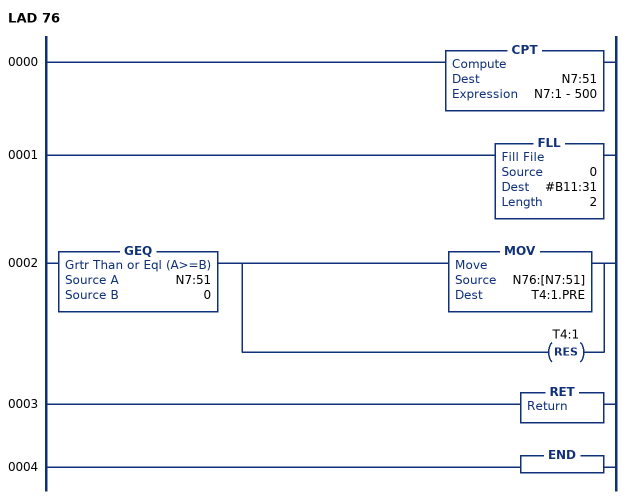
% Rung: 0 %
SOR CPT N7:51 " N7:1 - 500 " EOR
% Rung: 1 %
SOR FLL 0 #B11:31 2 EOR
% Rung: 2 %
SOR GEQ N7:51 0 BST MOV N76:[N7:51] T4:1.PRE NXB RES T4:1 BND EOR
% Rung: 3 %
SOR RET EOR
% Rung: 4 %
SOR END EOR

LADDER 77
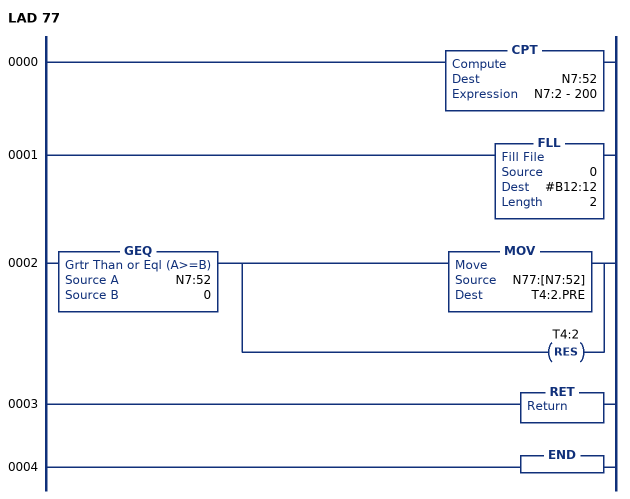
% Rung: 0 %
SOR CPT N7:52 " N7:2 - 200 " EOR
% Rung: 1 %
SOR FLL 0 #B12:12 2 EOR
% Rung: 2 %
SOR GEQ N7:52 0 BST MOV N77:[N7:52] T4:2.PRE NXB RES T4:2 BND EOR
% Rung: 3 %
SOR RET EOR
% Rung: 4 %
SOR END EOR

LADDER 78
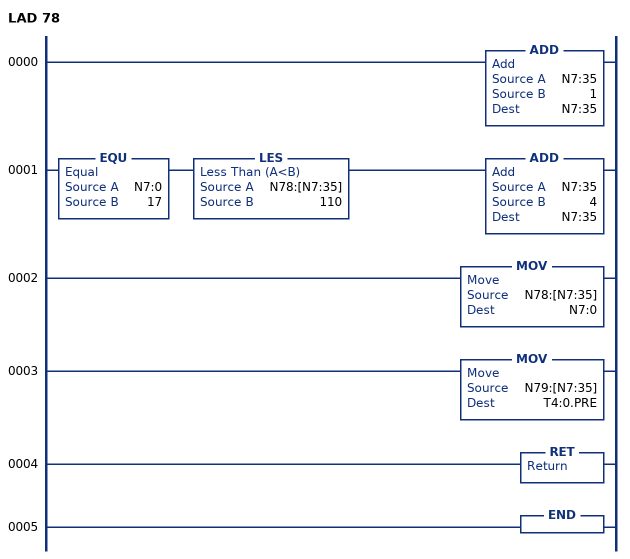
% Rung: 0 %
SOR ADD N7:35 1 N7:35 EOR
% Rung: 1 %
SOR EQU N7:0 17 LES N78:[N7:35] 110 ADD N7:35 4 N7:35 EOR
% Rung: 2 %
SOR MOV N78:[N7:35] N7:0 EOR
% Rung: 3 %
SOR MOV N79:[N7:35] T4:0.PRE EOR
% Rung: 4 %
SOR RET EOR
% Rung: 5 %
SOR END EOR

LADDER 80
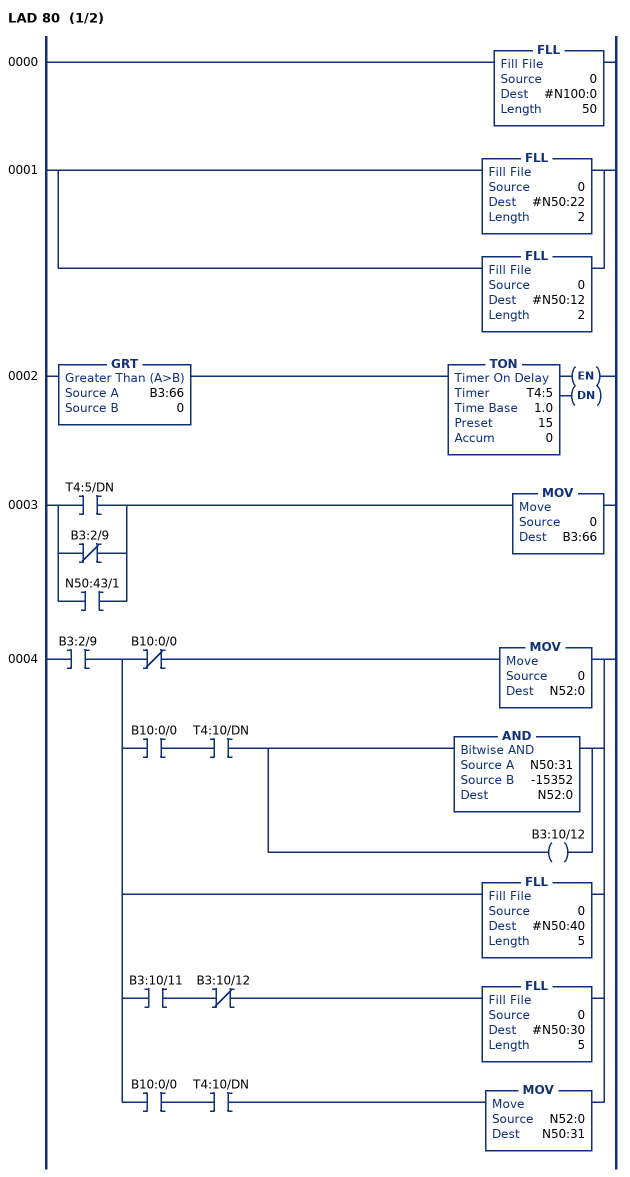
% Rung: 0 %
SOR FLL 0 #N100:0 50 EOR
% Rung: 1 %
SOR BST FLL 0 #N50:22 2 NXB FLL 0 #N50:12 2 BND EOR
% Rung: 2 %
SOR GRT B3:66 0 TON T4:5 1.0 15 0 EOR
% Rung: 3 %
SOR BST XIC T4:5/DN NXB XIO B3:2/9 NXB XIC N50:43/1 BND MOV 0 B3:66 EOR
% Rung: 4 %
SOR XIC B3:2/9 BST XIO B10:0/0 MOV 0 N52:0 NXB XIC B10:0/0 XIC T4:10/DN BST AND N50:31 -15352 N52:0 NXB OTE B3:10/12 BND NXB BST FLL 0 #N50:40 5 NXB XIC B3:10/11 XIO B3:10/12 FLL 0 #N50:30 5 BND NXB XIC B10:0/0 XIC T4:10/DN MOV N52:0 N50:31 BND EOR

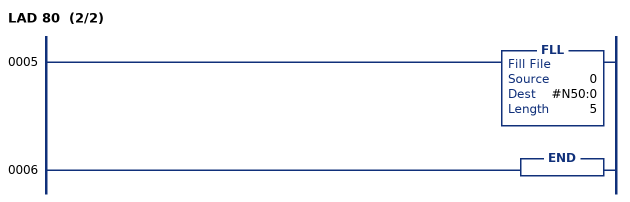
% Rung: 5 %
SOR FLL 0 #N50:0 5 EOR
% Rung: 6 %
SOR END EOR

LADDER 120
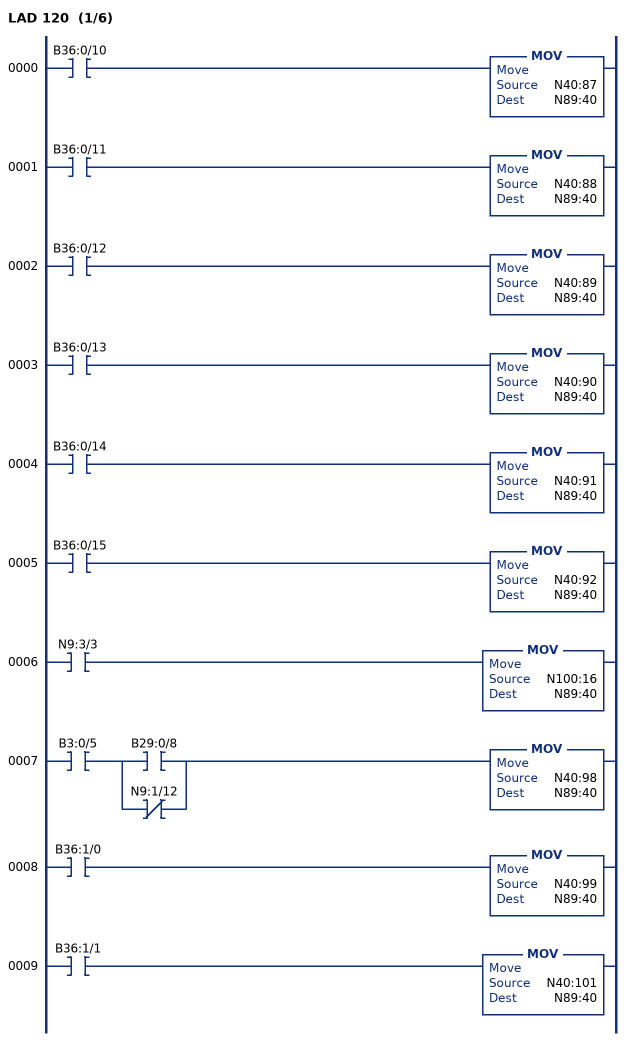
% Rung: 0 %
SOR XIC B36:0/10 MOV N40:87 N89:40 EOR
% Rung: 1 %
SOR XIC B36:0/11 MOV N40:88 N89:40 EOR
% Rung: 2 %
SOR XIC B36:0/12 MOV N40:89 N89:40 EOR
% Rung: 3 %
SOR XIC B36:0/13 MOV N40:90 N89:40 EOR
% Rung: 4 %
SOR XIC B36:0/14 MOV N40:91 N89:40 EOR
% Rung: 5 %
SOR XIC B36:0/15 MOV N40:92 N89:40 EOR
% Rung: 6 %
SOR XIC N9:3/3 MOV N100:16 N89:40 EOR
% Rung: 7 %
SOR XIC B3:0/5 BST XIC B29:0/8 NXB XIO N9:1/12 BND MOV N40:98 N89:40 EOR
% Rung: 8 %
SOR XIC B36:1/0 MOV N40:99 N89:40 EOR
% Rung: 9 %
SOR XIC B36:1/1 MOV N40:101 N89:40 EOR

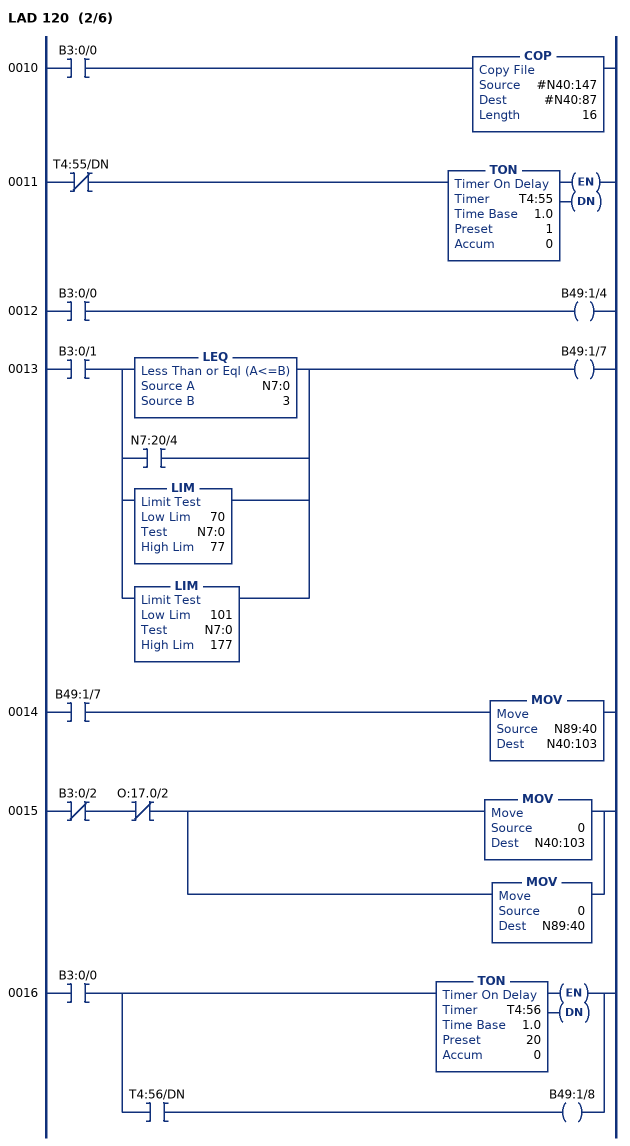
% Rung: 10 %
SOR XIC B3:0/0 COP #N40:147 #N40:87 16 EOR
% Rung: 11 %
SOR XIO T4:55/DN TON T4:55 1.0 1 0 EOR
% Rung: 12 %
SOR XIC B3:0/0 OTE B49:1/4 EOR
% Rung: 13 %
SOR XIC B3:0/1 BST LEQ N7:0 3 NXB XIC N7:20/4 NXB LIM 70 N7:0 77 NXB LIM 101 N7:0 177 BND OTE B49:1/7 EOR
% Rung: 14 %
SOR XIC B49:1/7 MOV N89:40 N40:103 EOR
% Rung: 15 %
SOR XIO B3:0/2 XIO O:17.0/2 BST MOV 0 N40:103 NXB MOV 0 N89:40 BND EOR
% Rung: 16 %
SOR XIC B3:0/0 BST TON T4:56 1.0 20 0 NXB XIC T4:56/DN OTE B49:1/8 BND EOR

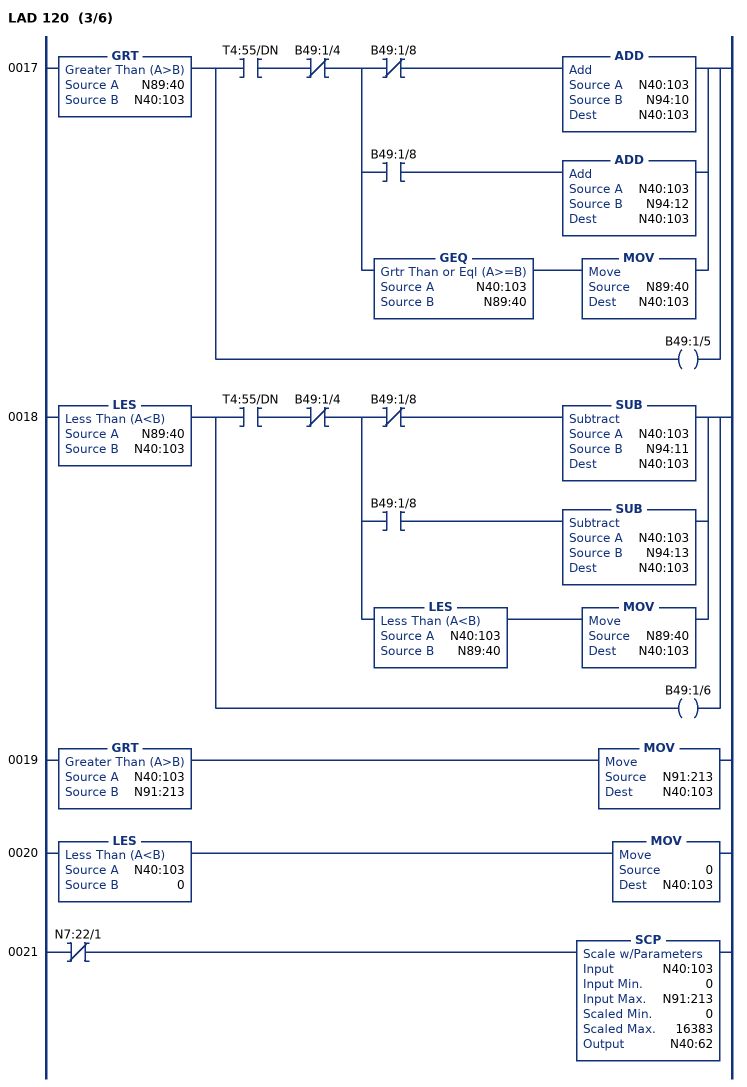
% Rung: 17 %
SOR GRT N89:40 N40:103 BST XIC T4:55/DN XIO B49:1/4 BST BST XIO B49:1/8 ADD N40:103 N94:10 N40:103 NXB XIC B49:1/8 ADD N40:103 N94:12 N40:103 BND NXB GEQ N40:103 N89:40 MOV N89:40 N40:103 BND NXB OTE B49:1/5 BND EOR
% Rung: 18 %
SOR LES N89:40 N40:103 BST XIC T4:55/DN XIO B49:1/4 BST BST XIO B49:1/8 SUB N40:103 N94:11 N40:103 NXB XIC B49:1/8 SUB N40:103 N94:13 N40:103 BND NXB LES N40:103 N89:40 MOV N89:40 N40:103 BND NXB OTE B49:1/6 BND EOR
% Rung: 19 %
SOR GRT N40:103 N91:213 MOV N91:213 N40:103 EOR
% Rung: 20 %
SOR LES N40:103 0 MOV 0 N40:103 EOR
% Rung: 21 %
SOR XIO N7:22/1 SCP N40:103 0 N91:213 0 16383 N40:62 EOR

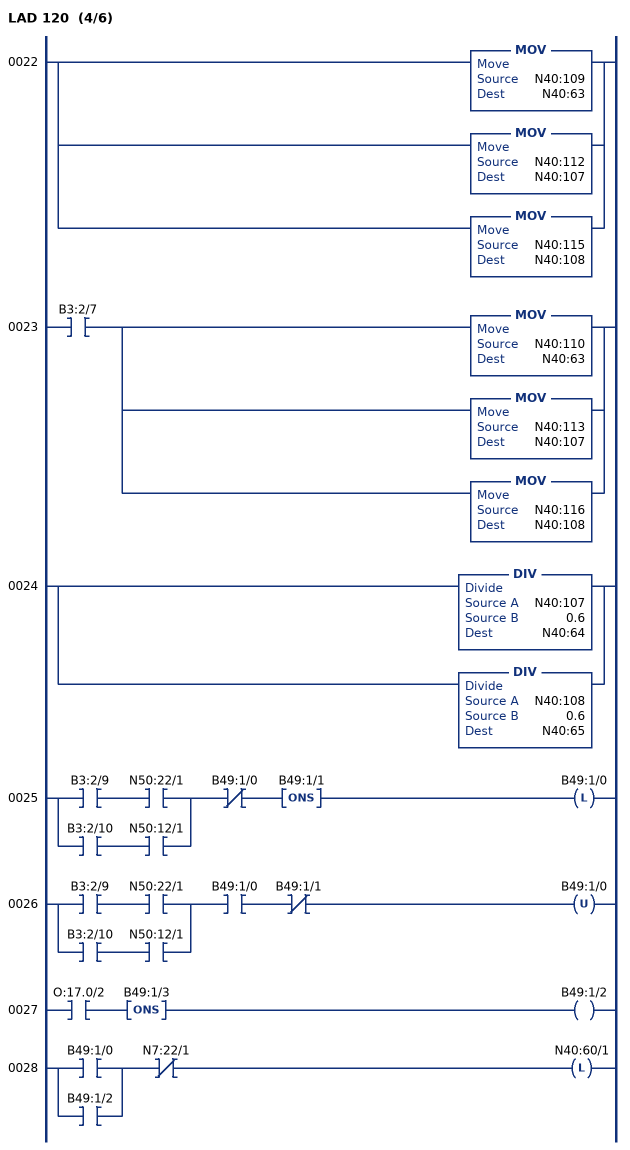
% Rung: 22 %
SOR BST MOV N40:109 N40:63 NXB MOV N40:112 N40:107 NXB MOV N40:115 N40:108 BND EOR
% Rung: 23 %
SOR XIC B3:2/7 BST MOV N40:110 N40:63 NXB MOV N40:113 N40:107 NXB MOV N40:116 N40:108 BND EOR
% Rung: 24 %
SOR BST DIV N40:107 0.6 N40:64 NXB DIV N40:108 0.6 N40:65 BND EOR
% Rung: 25 %
SOR BST XIC B3:2/9 XIC N50:22/1 NXB XIC B3:2/10 XIC N50:12/1 BND XIO B49:1/0 OSR B49:1/1 OTL B49:1/0 EOR
% Rung: 26 %
SOR BST XIC B3:2/9 XIC N50:22/1 NXB XIC B3:2/10 XIC N50:12/1 BND XIC B49:1/0 XIO B49:1/1 OTU B49:1/0 EOR
% Rung: 27 %
SOR XIC O:17.0/2 OSR B49:1/3 OTE B49:1/2 EOR
% Rung: 28 %
SOR BST XIC B49:1/0 NXB XIC B49:1/2 BND XIO N7:22/1 OTL N40:60/1 EOR

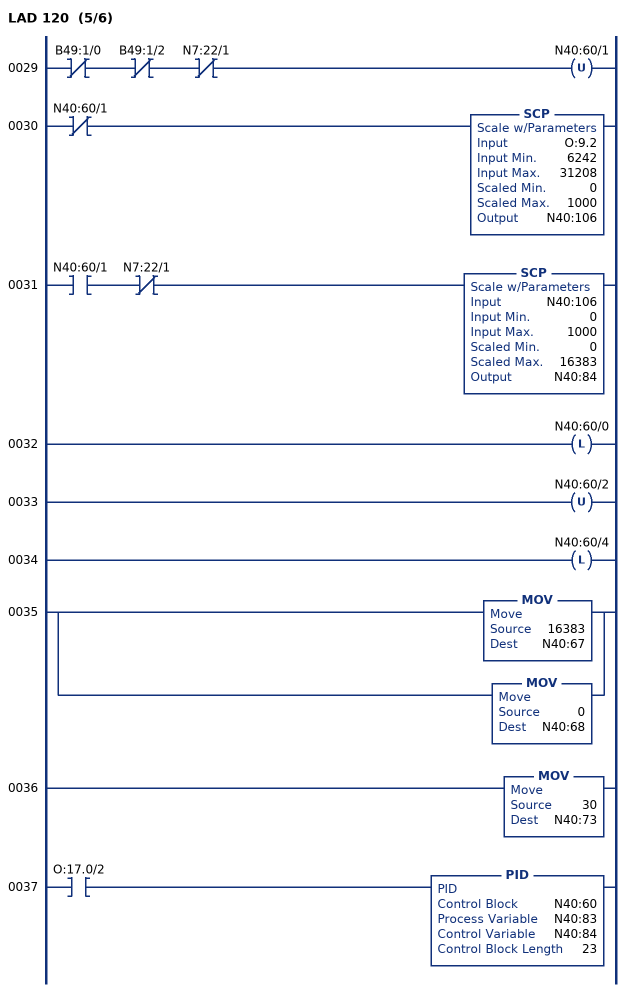
% Rung: 29 %
SOR XIO B49:1/0 XIO B49:1/2 XIO N7:22/1 OTU N40:60/1 EOR
% Rung: 30 %
SOR XIO N40:60/1 SCP O:9.2 6242 31208 0 1000 N40:106 EOR
% Rung: 31 %
SOR XIC N40:60/1 XIO N7:22/1 SCP N40:106 0 1000 0 16383 N40:84 EOR
% Rung: 32 %
SOR OTL N40:60/0 EOR
% Rung: 33 %
SOR OTU N40:60/2 EOR
% Rung: 34 %
SOR OTL N40:60/4 EOR
% Rung: 35 %
SOR BST MOV 16383 N40:67 NXB MOV 0 N40:68 BND EOR
% Rung: 36 %
SOR MOV 30 N40:73 EOR
% Rung: 37 %
SOR XIC O:17.0/2 PID N40:60 N40:83 N40:84 23 EOR

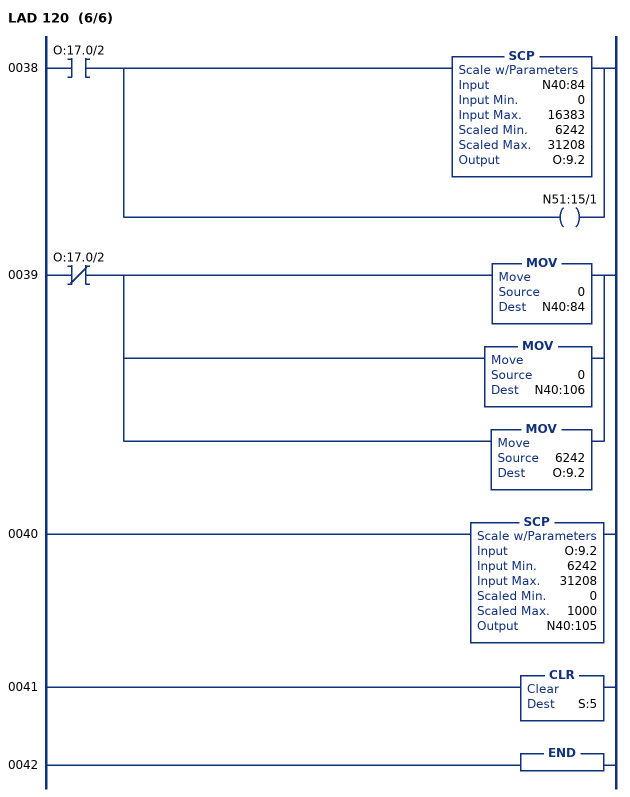
% Rung: 38 %
SOR XIC O:17.0/2 BST SCP N40:84 0 16383 6242 31208 O:9.2 NXB OTE N51:15/1 BND EOR
% Rung: 39 %
SOR XIO O:17.0/2 BST MOV 0 N40:84 NXB MOV 0 N40:106 NXB MOV 6242 O:9.2 BND EOR
% Rung: 40 %
SOR SCP O:9.2 6242 31208 0 1000 N40:105 EOR
% Rung: 41 %
SOR CLR S:5 EOR
% Rung: 42 %
SOR END EOR

LADDER 126
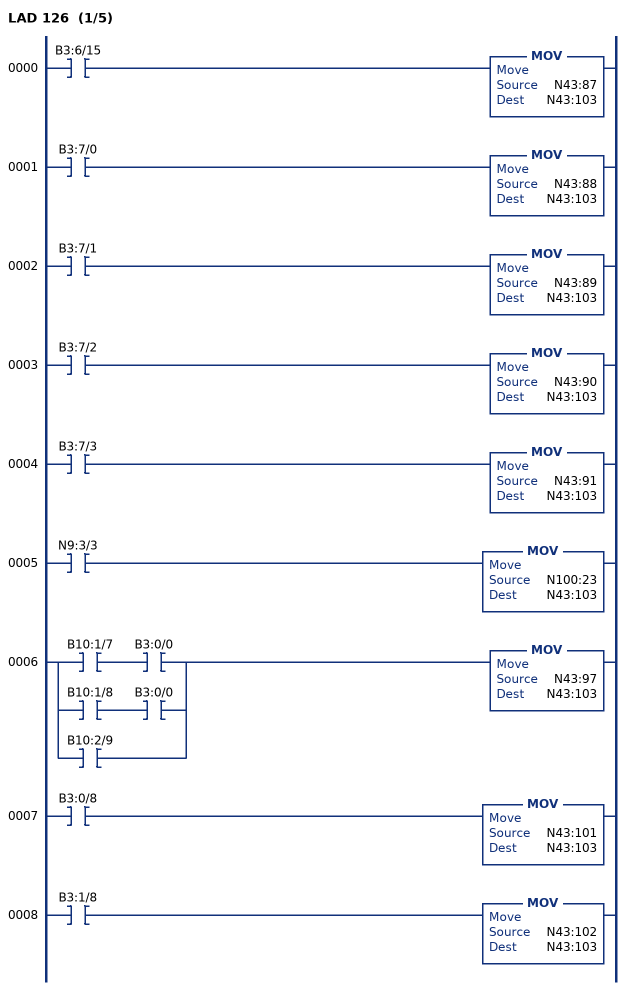
% Rung: 0 %
SOR XIC B3:6/15 MOV N43:87 N43:103 EOR
% Rung: 1 %
SOR XIC B3:7/0 MOV N43:88 N43:103 EOR
% Rung: 2 %
SOR XIC B3:7/1 MOV N43:89 N43:103 EOR
% Rung: 3 %
SOR XIC B3:7/2 MOV N43:90 N43:103 EOR
% Rung: 4 %
SOR XIC B3:7/3 MOV N43:91 N43:103 EOR
% Rung: 5 %
SOR XIC N9:3/3 MOV N100:23 N43:103 EOR
% Rung: 6 %
SOR BST XIC B10:1/7 XIC B3:0/0 NXB XIC B10:1/8 XIC B3:0/0 NXB XIC B10:2/9 BND MOV N43:97 N43:103 EOR
% Rung: 7 %
SOR XIC B3:0/8 MOV N43:101 N43:103 EOR
% Rung: 8 %
SOR XIC B3:1/8 MOV N43:102 N43:103 EOR

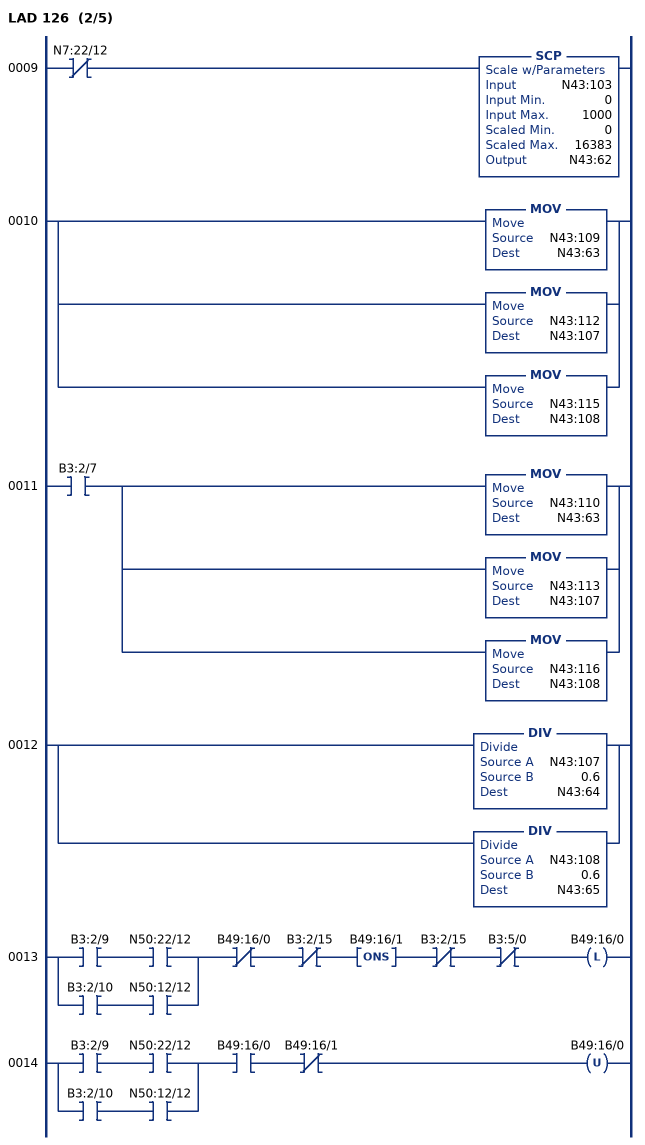
% Rung: 9 %
SOR XIO N7:22/12 SCP N43:103 0 1000 0 16383 N43:62 EOR
% Rung: 10 %
SOR BST MOV N43:109 N43:63 NXB MOV N43:112 N43:107 NXB MOV N43:115 N43:108 BND EOR
% Rung: 11 %
SOR XIC B3:2/7 BST MOV N43:110 N43:63 NXB MOV N43:113 N43:107 NXB MOV N43:116 N43:108 BND EOR
% Rung: 12 %
SOR BST DIV N43:107 0.6 N43:64 NXB DIV N43:108 0.6 N43:65 BND EOR
% Rung: 13 %
SOR BST XIC B3:2/9 XIC N50:22/12 NXB XIC B3:2/10 XIC N50:12/12 BND XIO B49:16/0 XIO B3:2/15 OSR B49:16/1 XIO B3:2/15 XIO B3:5/0 OTL B49:16/0 EOR
% Rung: 14 %
SOR BST XIC B3:2/9 XIC N50:22/12 NXB XIC B3:2/10 XIC N50:12/12 BND XIC B49:16/0 XIO B49:16/1 OTU B49:16/0 EOR

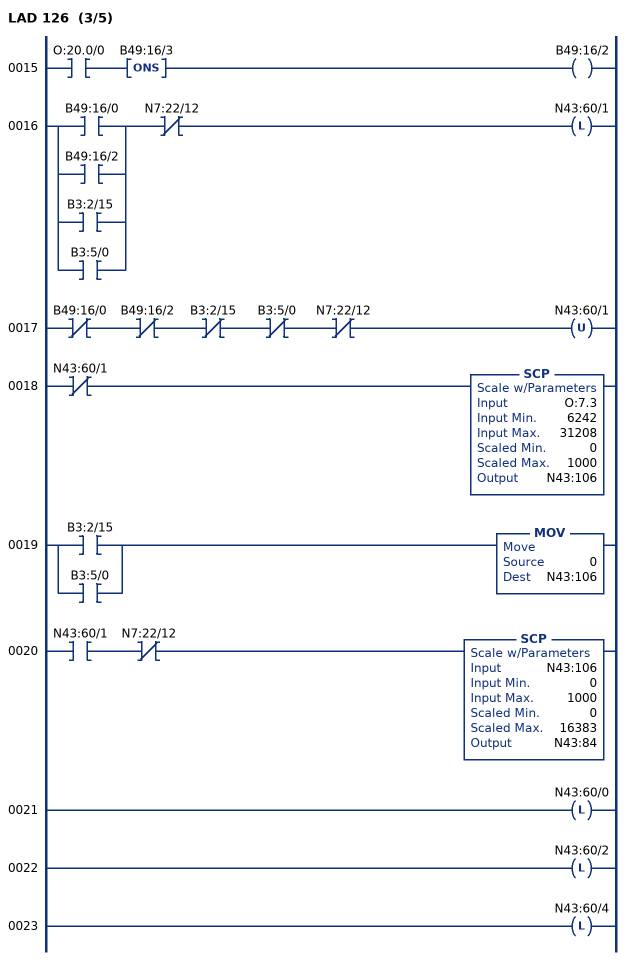
% Rung: 15 %
SOR XIC O:20.0/0 OSR B49:16/3 OTE B49:16/2 EOR
% Rung: 16 %
SOR BST XIC B49:16/0 NXB XIC B49:16/2 NXB XIC B3:2/15 NXB XIC B3:5/0 BND XIO N7:22/12 OTL N43:60/1 EOR
% Rung: 17 %
SOR XIO B49:16/0 XIO B49:16/2 XIO B3:2/15 XIO B3:5/0 XIO N7:22/12 OTU N43:60/1 EOR
% Rung: 18 %
SOR XIO N43:60/1 SCP O:7.3 6242 31208 0 1000 N43:106 EOR
% Rung: 19 %
SOR BST XIC B3:2/15 NXB XIC B3:5/0 BND MOV 0 N43:106 EOR
% Rung: 20 %
SOR XIC N43:60/1 XIO N7:22/12 SCP N43:106 0 1000 0 16383 N43:84 EOR
% Rung: 21 %
SOR OTL N43:60/0 EOR
% Rung: 22 %
SOR OTL N43:60/2 EOR
% Rung: 23 %
SOR OTL N43:60/4 EOR

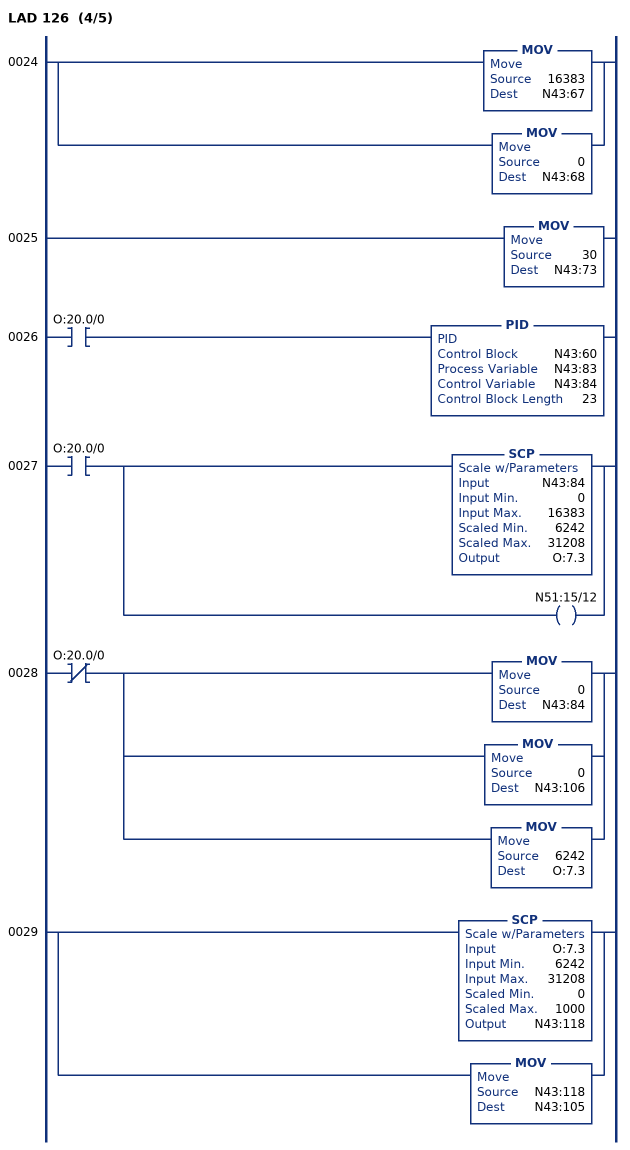
% Rung: 24 %
SOR BST MOV 16383 N43:67 NXB MOV 0 N43:68 BND EOR
% Rung: 25 %
SOR MOV 30 N43:73 EOR
% Rung: 26 %
SOR XIC O:20.0/0 PID N43:60 N43:83 N43:84 23 EOR
% Rung: 27 %
SOR XIC O:20.0/0 BST SCP N43:84 0 16383 6242 31208 O:7.3 NXB OTE N51:15/12 BND EOR
% Rung: 28 %
SOR XIO O:20.0/0 BST MOV 0 N43:84 NXB MOV 0 N43:106 NXB MOV 6242 O:7.3 BND EOR
% Rung: 29 %
SOR BST SCP O:7.3 6242 31208 0 1000 N43:118 NXB MOV N43:118 N43:105 BND EOR

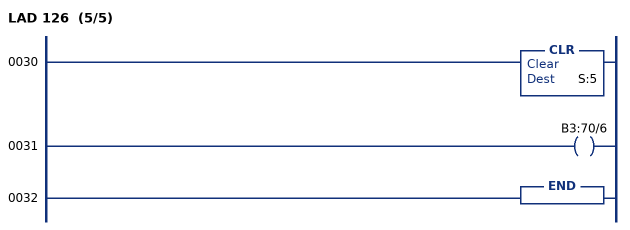
% Rung: 30 %
SOR CLR S:5 EOR
% Rung: 31 %
SOR OTE B3:70/6 EOR
% Rung: 32 %
SOR END EOR

LADDER 127
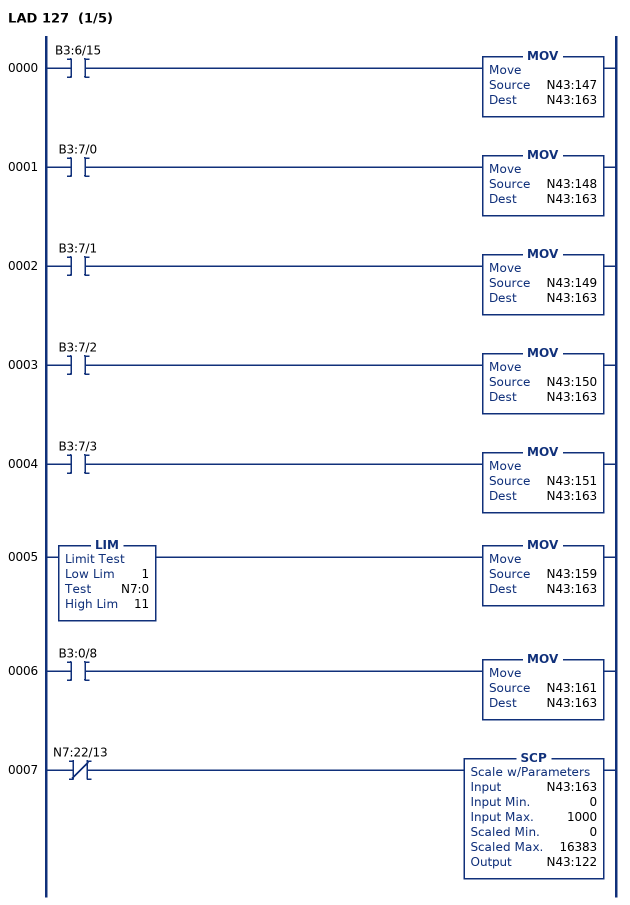
% Rung: 0 %
SOR XIC B3:6/15 MOV N43:147 N43:163 EOR
% Rung: 1 %
SOR XIC B3:7/0 MOV N43:148 N43:163 EOR
% Rung: 2 %
SOR XIC B3:7/1 MOV N43:149 N43:163 EOR
% Rung: 3 %
SOR XIC B3:7/2 MOV N43:150 N43:163 EOR
% Rung: 4 %
SOR XIC B3:7/3 MOV N43:151 N43:163 EOR
% Rung: 5 %
SOR LIM 1 N7:0 11 MOV N43:159 N43:163 EOR
% Rung: 6 %
SOR XIC B3:0/8 MOV N43:161 N43:163 EOR
% Rung: 7 %
SOR XIO N7:22/13 SCP N43:163 0 1000 0 16383 N43:122 EOR

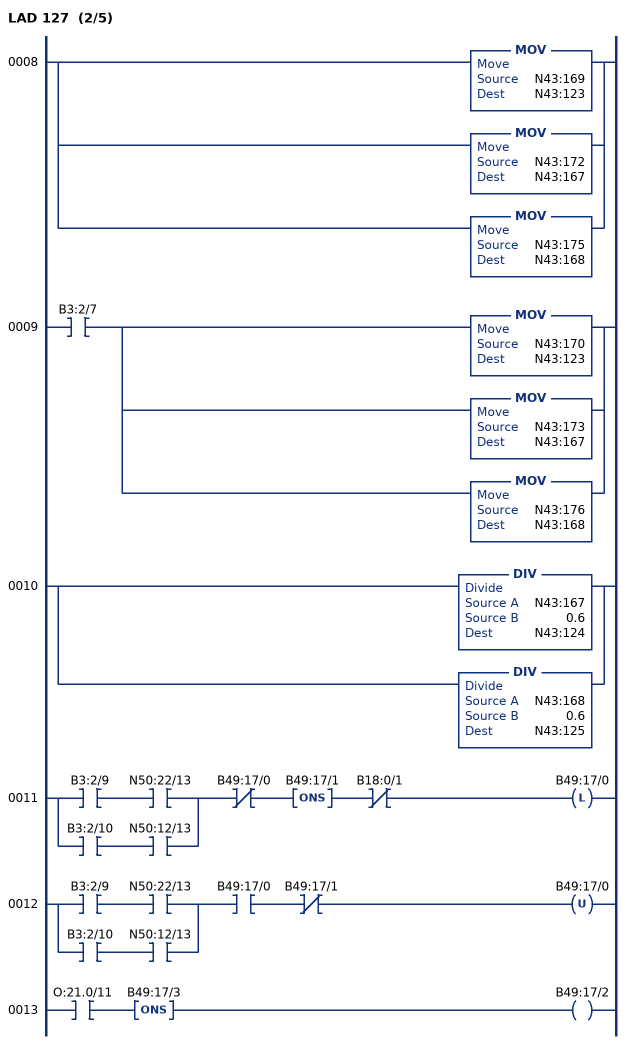
% Rung: 8 %
SOR BST MOV N43:169 N43:123 NXB MOV N43:172 N43:167 NXB MOV N43:175 N43:168 BND EOR
% Rung: 9 %
SOR XIC B3:2/7 BST MOV N43:170 N43:123 NXB MOV N43:173 N43:167 NXB MOV N43:176 N43:168 BND EOR
% Rung: 10 %
SOR BST DIV N43:167 0.6 N43:124 NXB DIV N43:168 0.6 N43:125 BND EOR
% Rung: 11 %
SOR BST XIC B3:2/9 XIC N50:22/13 NXB XIC B3:2/10 XIC N50:12/13 BND XIO B49:17/0 OSR B49:17/1 XIO B18:0/1 OTL B49:17/0 EOR
% Rung: 12 %
SOR BST XIC B3:2/9 XIC N50:22/13 NXB XIC B3:2/10 XIC N50:12/13 BND XIC B49:17/0 XIO B49:17/1 OTU B49:17/0 EOR
% Rung: 13 %
SOR XIC O:21.0/11 OSR B49:17/3 OTE B49:17/2 EOR

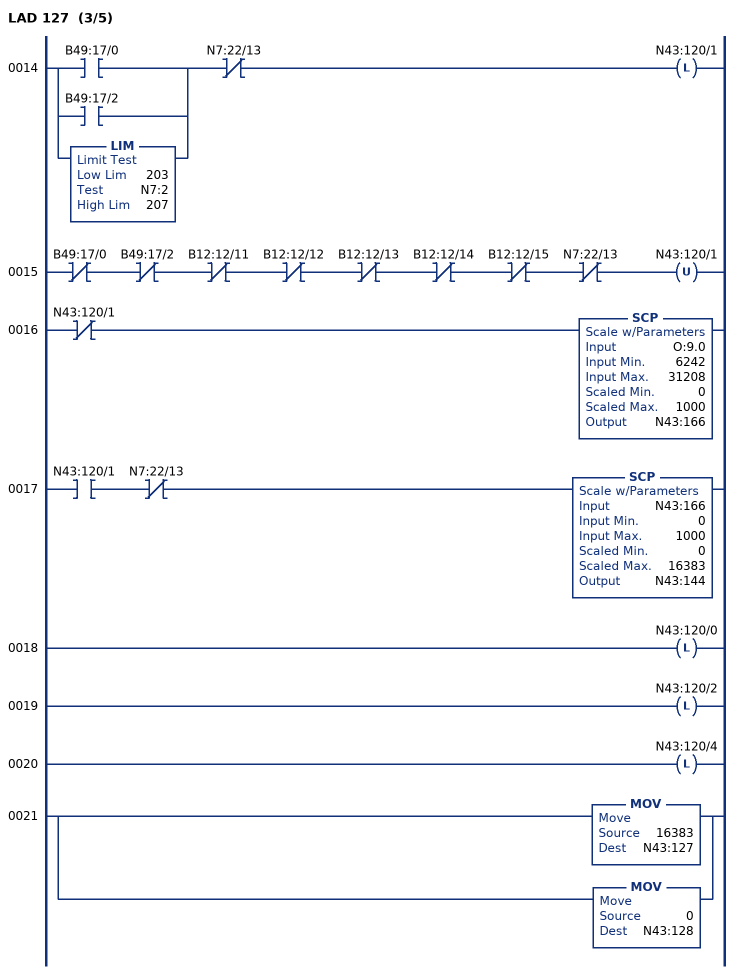
% Rung: 14 %
SOR BST XIC B49:17/0 NXB XIC B49:17/2 NXB LIM 203 N7:2 207 BND XIO N7:22/13 OTL N43:120/1 EOR
% Rung: 15 %
SOR XIO B49:17/0 XIO B49:17/2 XIO B12:12/11 XIO B12:12/12 XIO B12:12/13 XIO B12:12/14 XIO B12:12/15 XIO N7:22/13 OTU N43:120/1 EOR
% Rung: 16 %
SOR XIO N43:120/1 SCP O:9.0 6242 31208 0 1000 N43:166 EOR
% Rung: 17 %
SOR XIC N43:120/1 XIO N7:22/13 SCP N43:166 0 1000 0 16383 N43:144 EOR
% Rung: 18 %
SOR OTL N43:120/0 EOR
% Rung: 19 %
SOR OTL N43:120/2 EOR
% Rung: 20 %
SOR OTL N43:120/4 EOR
% Rung: 21 %
SOR BST MOV 16383 N43:127 NXB MOV 0 N43:128 BND EOR

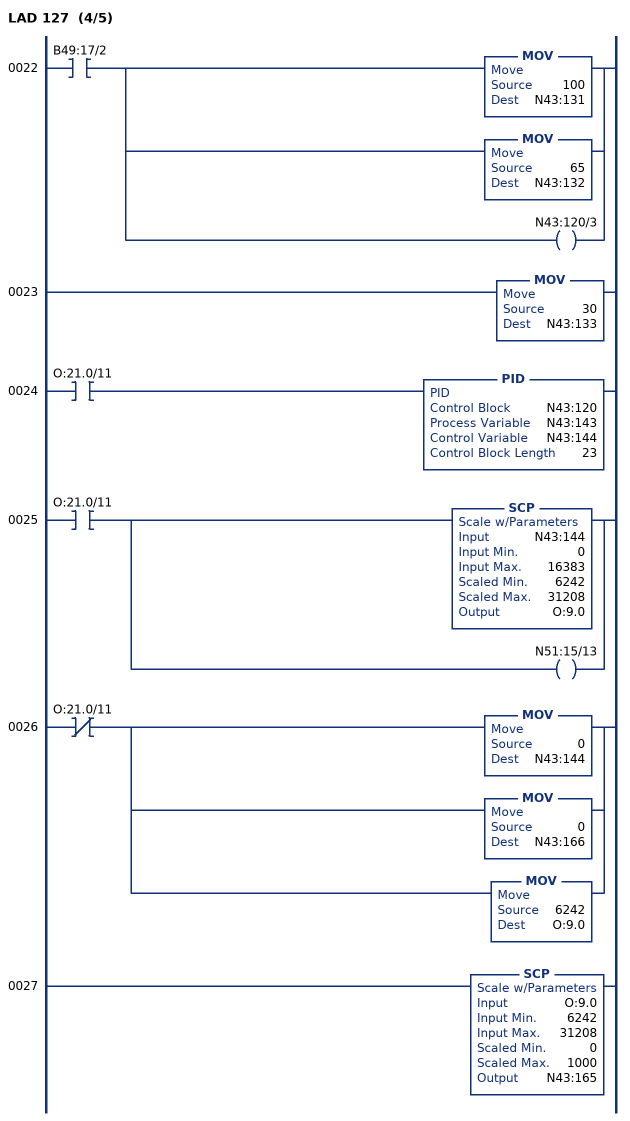
% Rung: 22 %
SOR XIC B49:17/2 BST MOV 100 N43:131 NXB MOV 65 N43:132 NXB OTE N43:120/3 BND EOR
% Rung: 23 %
SOR MOV 30 N43:133 EOR
% Rung: 24 %
SOR XIC O:21.0/11 PID N43:120 N43:143 N43:144 23 EOR
% Rung: 25 %
SOR XIC O:21.0/11 BST SCP N43:144 0 16383 6242 31208 O:9.0 NXB OTE N51:15/13 BND EOR
% Rung: 26 %
SOR XIO O:21.0/11 BST MOV 0 N43:144 NXB MOV 0 N43:166 NXB MOV 6242 O:9.0 BND EOR
% Rung: 27 %
SOR SCP O:9.0 6242 31208 0 1000 N43:165 EOR

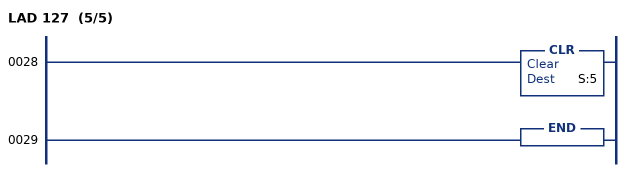
% Rung: 28 %
SOR CLR S:5 EOR
% Rung: 29 %
SOR END EOR

LADDER 129
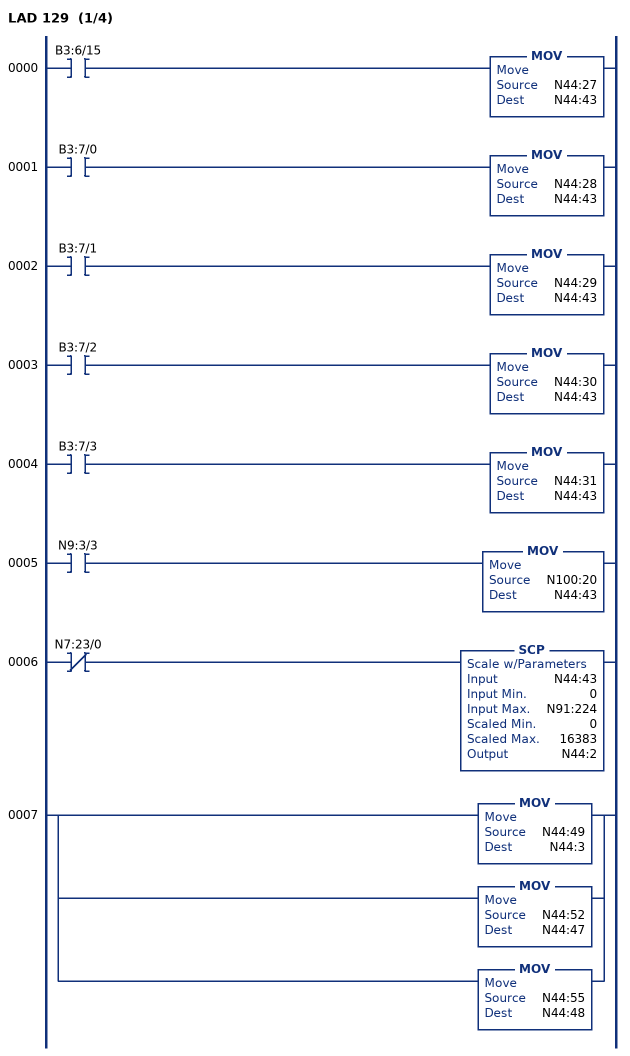
% Rung: 0 %
SOR XIC B3:6/15 MOV N44:27 N44:43 EOR
% Rung: 1 %
SOR XIC B3:7/0 MOV N44:28 N44:43 EOR
% Rung: 2 %
SOR XIC B3:7/1 MOV N44:29 N44:43 EOR
% Rung: 3 %
SOR XIC B3:7/2 MOV N44:30 N44:43 EOR
% Rung: 4 %
SOR XIC B3:7/3 MOV N44:31 N44:43 EOR
% Rung: 5 %
SOR XIC N9:3/3 MOV N100:20 N44:43 EOR
% Rung: 6 %
SOR XIO N7:23/0 SCP N44:43 0 N91:224 0 16383 N44:2 EOR
% Rung: 7 %
SOR BST MOV N44:49 N44:3 NXB MOV N44:52 N44:47 NXB MOV N44:55 N44:48 BND EOR

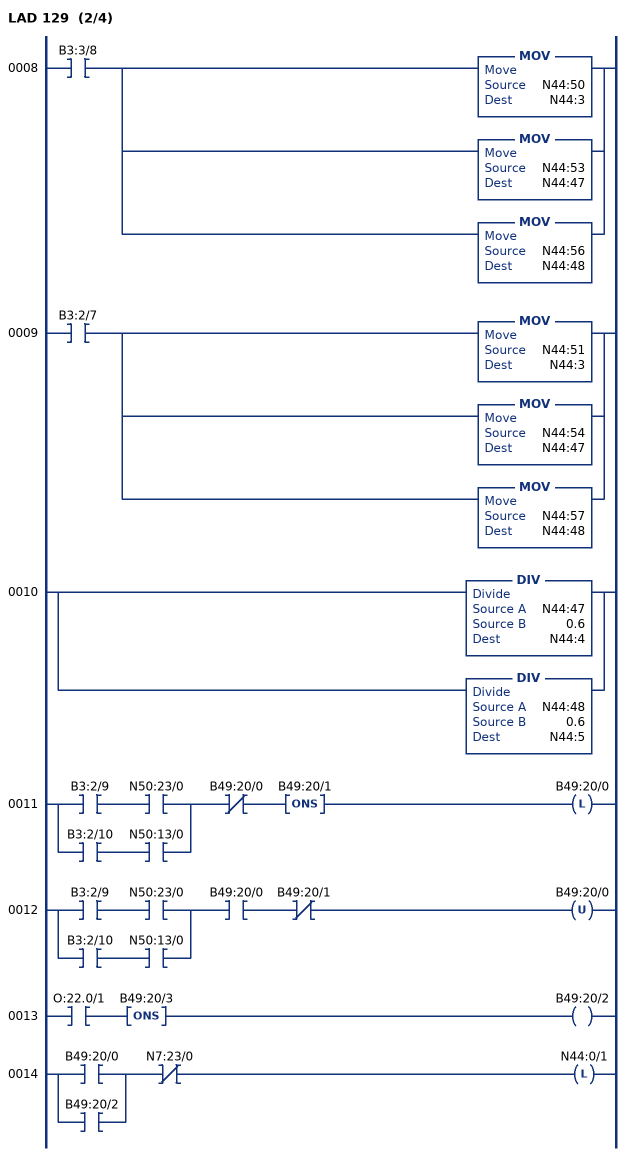
% Rung: 8 %
SOR XIC B3:3/8 BST MOV N44:50 N44:3 NXB MOV N44:53 N44:47 NXB MOV N44:56 N44:48 BND EOR
% Rung: 9 %
SOR XIC B3:2/7 BST MOV N44:51 N44:3 NXB MOV N44:54 N44:47 NXB MOV N44:57 N44:48 BND EOR
% Rung: 10 %
SOR BST DIV N44:47 0.6 N44:4 NXB DIV N44:48 0.6 N44:5 BND EOR
% Rung: 11 %
SOR BST XIC B3:2/9 XIC N50:23/0 NXB XIC B3:2/10 XIC N50:13/0 BND XIO B49:20/0 OSR B49:20/1 OTL B49:20/0 EOR
% Rung: 12 %
SOR BST XIC B3:2/9 XIC N50:23/0 NXB XIC B3:2/10 XIC N50:13/0 BND XIC B49:20/0 XIO B49:20/1 OTU B49:20/0 EOR
% Rung: 13 %
SOR XIC O:22.0/1 OSR B49:20/3 OTE B49:20/2 EOR
% Rung: 14 %
SOR BST XIC B49:20/0 NXB XIC B49:20/2 BND XIO N7:23/0 OTL N44:0/1 EOR

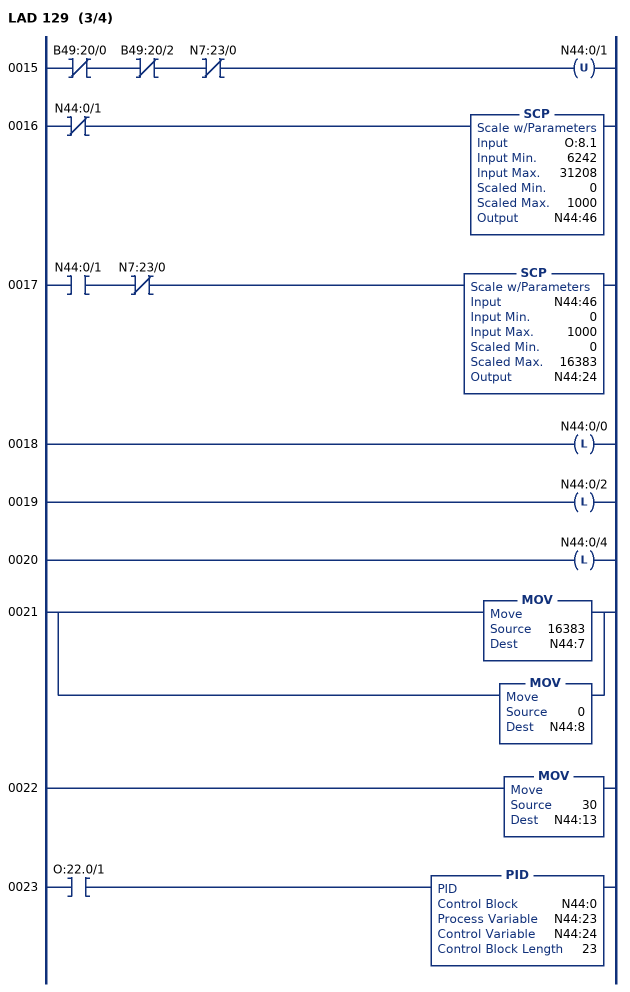
% Rung: 15 %
SOR XIO B49:20/0 XIO B49:20/2 XIO N7:23/0 OTU N44:0/1 EOR
% Rung: 16 %
SOR XIO N44:0/1 SCP O:8.1 6242 31208 0 1000 N44:46 EOR
% Rung: 17 %
SOR XIC N44:0/1 XIO N7:23/0 SCP N44:46 0 1000 0 16383 N44:24 EOR
% Rung: 18 %
SOR OTL N44:0/0 EOR
% Rung: 19 %
SOR OTL N44:0/2 EOR
% Rung: 20 %
SOR OTL N44:0/4 EOR
% Rung: 21 %
SOR BST MOV 16383 N44:7 NXB MOV 0 N44:8 BND EOR
% Rung: 22 %
SOR MOV 30 N44:13 EOR
% Rung: 23 %
SOR XIC O:22.0/1 PID N44:0 N44:23 N44:24 23 EOR

